PROGRAM Axis01_Manual
VAR
//System_Bit
	Always_ON	:	BOOL	:=TRUE	;//상시 ON 
	Always_OFF	:	BOOL	:=FALSE	;//상시 OFF
END_VAR
VAR // added by the converter: edge detectors and wires of the graphical bodies
    _rt1, _rt2, _rt3 : R_TRIG;
END_VAR

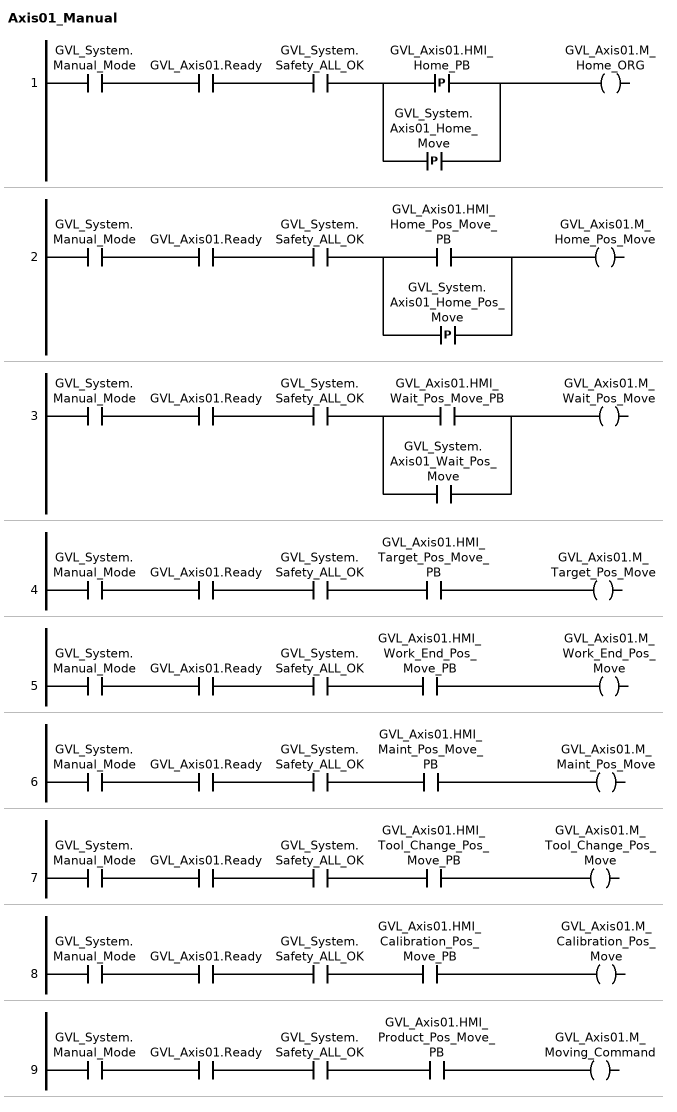
// NETWORK 1
_rt1(CLK := GVL_Axis01.HMI_Home_PB);
_rt2(CLK := GVL_System.Axis01_Home_Move);
GVL_Axis01.M_Home_ORG := GVL_System.Manual_Mode AND GVL_Axis01.Ready AND GVL_System.Safety_ALL_OK AND (_rt1.Q OR _rt2.Q);

// NETWORK 2
_rt3(CLK := GVL_System.Axis01_Home_Pos_Move);
GVL_Axis01.M_Home_Pos_Move := GVL_System.Manual_Mode AND GVL_Axis01.Ready AND GVL_System.Safety_ALL_OK AND (GVL_Axis01.HMI_Home_Pos_Move_PB OR _rt3.Q);

// NETWORK 3
GVL_Axis01.M_Wait_Pos_Move := GVL_System.Manual_Mode AND GVL_Axis01.Ready AND GVL_System.Safety_ALL_OK AND (GVL_Axis01.HMI_Wait_Pos_Move_PB OR GVL_System.Axis01_Wait_Pos_Move);

// NETWORK 4
GVL_Axis01.M_Target_Pos_Move := GVL_System.Manual_Mode AND GVL_Axis01.Ready AND GVL_System.Safety_ALL_OK AND GVL_Axis01.HMI_Target_Pos_Move_PB;

// NETWORK 5
GVL_Axis01.M_Work_End_Pos_Move := GVL_System.Manual_Mode AND GVL_Axis01.Ready AND GVL_System.Safety_ALL_OK AND GVL_Axis01.HMI_Work_End_Pos_Move_PB;

// NETWORK 6
GVL_Axis01.M_Maint_Pos_Move := GVL_System.Manual_Mode AND GVL_Axis01.Ready AND GVL_System.Safety_ALL_OK AND GVL_Axis01.HMI_Maint_Pos_Move_PB;

// NETWORK 7
GVL_Axis01.M_Tool_Change_Pos_Move := GVL_System.Manual_Mode AND GVL_Axis01.Ready AND GVL_System.Safety_ALL_OK AND GVL_Axis01.HMI_Tool_Change_Pos_Move_PB;

// NETWORK 8
GVL_Axis01.M_Calibration_Pos_Move := GVL_System.Manual_Mode AND GVL_Axis01.Ready AND GVL_System.Safety_ALL_OK AND GVL_Axis01.HMI_Calibration_Pos_Move_PB;

// NETWORK 9
GVL_Axis01.M_Moving_Command := GVL_System.Manual_Mode AND GVL_Axis01.Ready AND GVL_System.Safety_ALL_OK AND GVL_Axis01.HMI_Product_Pos_Move_PB;

END_PROGRAM

(* stored: Version 1.1.0.1, ProductVersion 3.1.4024.15
   POU Axis01_Manual: Id {a5627c4c-9b0e-420c-ab5f-e3b931e0e900}, SpecialFunc None *)
